{attribute 'qualified_only'}
{attribute 'to_string'}
TYPE enum_FB_MON :
(
	undefine := 0,
	run :=1,
	stop :=2,
	safe :=3,
	error := 4,
	reset := 5,
	start := 6,
	errdelay := 7,
	delayout :=8,
	functest := 9
);
END_TYPE

(* stored: Version 1.1.0.1
   DUT enum_FB_MON: Id {79b6bdec-34e4-4a7f-8426-e4c650c43ef3} *)
